{attribute 'OPC.UA.DA.StructuredType' := '1'}
TYPE SConditionSpec :
STRUCT
	IsActive: BOOL;
	ExpressionType: EExpressionType;
	ExpressionIdx: UINT;
END_STRUCT
END_TYPE

(* stored: Version 1.1.0.1
   DUT SConditionSpec: Id {a5c224f8-bf2b-4baa-b19d-f999eca225a1} *)
